# EPICS StreamDevice protocol: jeonglee-DemoApp/Db/training.proto
sendRawQuery {
  ExtraInput = Ignore;
  out "%s";
  in  "%(\$1)40c";
}
